// TIA Portal V15.1 export
// export: Created 2020-06-12T07:35:42.5849609Z, ExportSetting None, DisplayName Totally Integrated Automation Portal, DisplayVersion V15.1, DisplayName TIA Portal Openness, DisplayVersion V15.1, DisplayName STEP 7 Professional, DisplayVersion V15.1, DisplayName STEP 7 Safety, DisplayVersion V15.1, DisplayName WinCC Advanced, DisplayVersion V15.1
FUNCTION "CW_Module" : Void   // FC118, FBD
TITLE = CW Module (HC-lines cooling) handle
{ S7_Optimized_Access := 'TRUE' }
// stored: SetENOAutomatically False
   VAR_TEMP
      tStart_heater : Bool;
      tHeater_on : Bool;
      pump1_start : Bool;
      pump2_start : Bool;
      _heat_off : Real;
      tReqOn : Bool;
      tReqOff : Bool;
      tStage : Int;
      tFlowset : Real;
      tCVMin : Real;
      tCVMax : Real;
   END_VAR
   VAR_TEMP   // added for the SCL form of the ladder/FBD networks
      _w1 : Bool;
      _w2 : Bool;
   END_VAR
BEGIN

REGION Network 1: HMI request treat
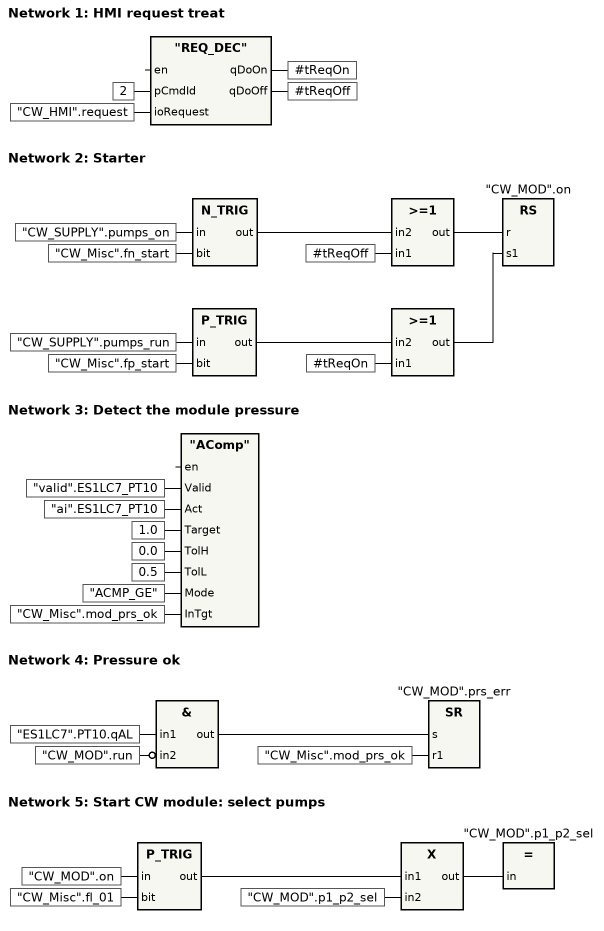
   "REQ_DEC"(pCmdId := 2, ioRequest := "CW_HMI".request, qDoOn => #tReqOn, qDoOff => #tReqOff);
END_REGION

REGION Network 2: Starter
   #_w1 := NOT "CW_SUPPLY".pumps_on AND "CW_Misc".fn_start;   // falling edge
   "CW_Misc".fn_start := "CW_SUPPLY".pumps_on;
   #_w2 := "CW_SUPPLY".pumps_run AND NOT "CW_Misc".fp_start;   // rising edge
   "CW_Misc".fp_start := "CW_SUPPLY".pumps_run;
   IF #_w1 OR #tReqOff THEN
       "CW_MOD".on := FALSE;   // RS flip-flop
   END_IF;
   IF #_w2 OR #tReqOn THEN "CW_MOD".on := TRUE; END_IF;
END_REGION

REGION Network 3: Detect the module pressure
   "AComp"(Valid := "valid".ES1LC7_PT10,
           Act := "ai".ES1LC7_PT10,
           Target := 1.0,
           TolH := 0.0,
           TolL := 0.5,
           Mode := "ACMP_GE",
           InTgt := "CW_Misc".mod_prs_ok);
END_REGION

REGION Network 4: Pressure ok
   // That is critical only before start
   IF "ES1LC7".PT10.qAL AND NOT "CW_MOD".run THEN
       "CW_MOD".prs_err := TRUE;   // SR flip-flop
   END_IF;
   IF "CW_Misc".mod_prs_ok THEN "CW_MOD".prs_err := FALSE; END_IF;
END_REGION

REGION Network 5: Start CW module: select pumps
   #_w1 := "CW_MOD".on AND NOT "CW_Misc".fl_01;   // rising edge
   "CW_Misc".fl_01 := "CW_MOD".on;
   "CW_MOD".p1_p2_sel := #_w1 XOR "CW_MOD".p1_p2_sel;
END_REGION

REGION Network 6: Module pumps LOCK
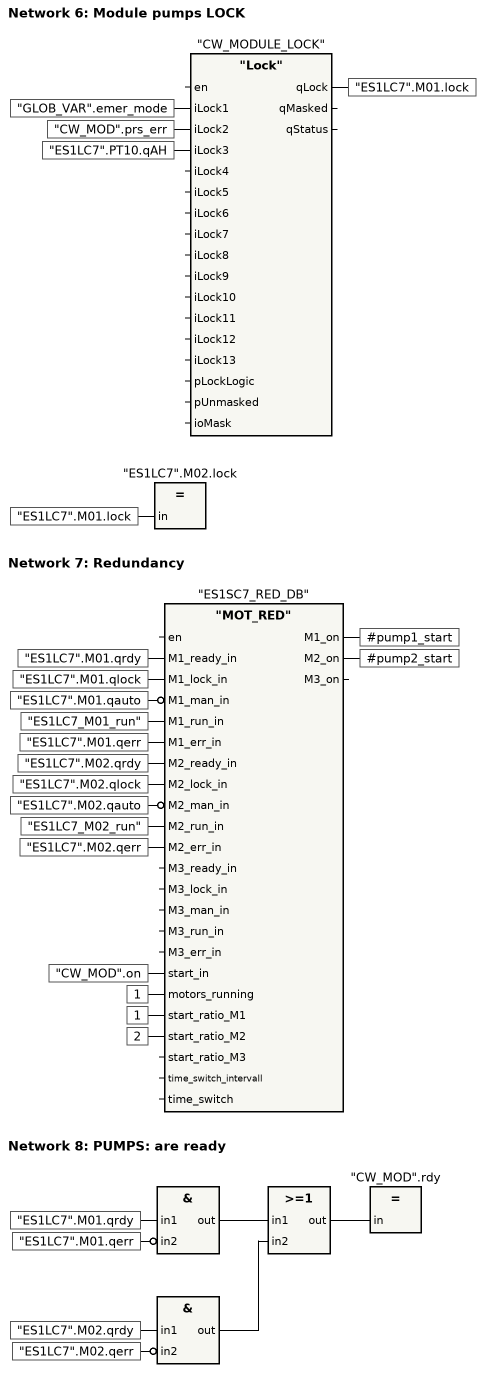
   "CW_MODULE_LOCK"(iLock1 := "GLOB_VAR".emer_mode,   // "Lock"
                    iLock2 := "CW_MOD".prs_err,
                    iLock3 := "ES1LC7".PT10.qAH,
                    qLock => "ES1LC7".M01.lock);
   "ES1LC7".M02.lock := "ES1LC7".M01.lock;
END_REGION

REGION Network 7: Redundancy
   "ES1SC7_RED_DB"(M1_ready_in := "ES1LC7".M01.qrdy,   // "MOT_RED"
                   M1_lock_in := "ES1LC7".M01.qlock,
                   M1_man_in := NOT "ES1LC7".M01.qauto,
                   M1_run_in := "ES1LC7_M01_run",
                   M1_err_in := "ES1LC7".M01.qerr,
                   M2_ready_in := "ES1LC7".M02.qrdy,
                   M2_lock_in := "ES1LC7".M02.qlock,
                   M2_man_in := NOT "ES1LC7".M02.qauto,
                   M2_run_in := "ES1LC7_M02_run",
                   M2_err_in := "ES1LC7".M02.qerr,
                   start_in := "CW_MOD".on,
                   motors_running := 1,
                   start_ratio_M1 := 1,
                   start_ratio_M2 := 2,
                   M1_on => #pump1_start,
                   M2_on => #pump2_start);
END_REGION

REGION Network 8: PUMPS: are ready
   "CW_MOD".rdy := ("ES1LC7".M01.qrdy AND NOT "ES1LC7".M01.qerr) OR ("ES1LC7".M02.qrdy AND NOT "ES1LC7".M02.qerr);
END_REGION

REGION Network 9: PUMPs: are(is) running
   // The stable running state is delayed for a ramp time.
   // In this case the ramp time is 50s, we take 60s.
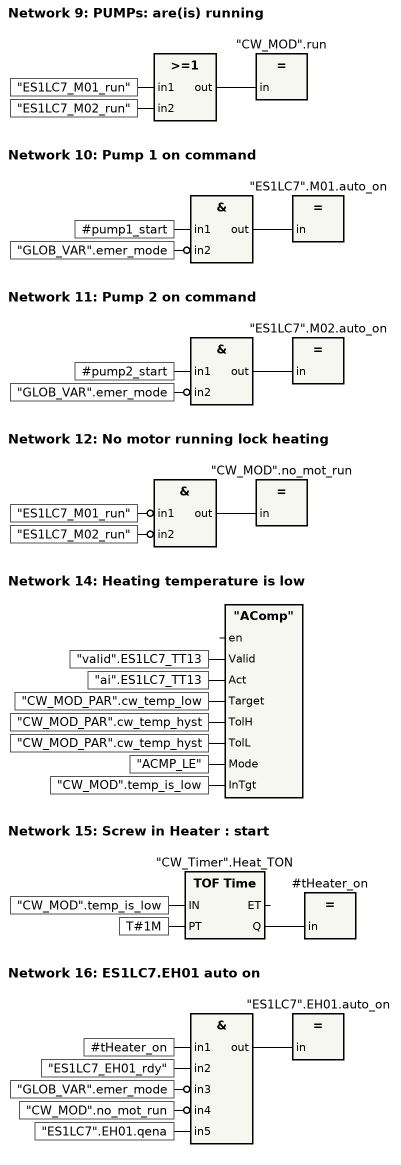
   "CW_MOD".run := "ES1LC7_M01_run" OR "ES1LC7_M02_run";
END_REGION

REGION Network 10: Pump 1 on command
   "ES1LC7".M01.auto_on := #pump1_start AND NOT "GLOB_VAR".emer_mode;
END_REGION

REGION Network 11: Pump 2 on command
   "ES1LC7".M02.auto_on := #pump2_start AND NOT "GLOB_VAR".emer_mode;
END_REGION

REGION Network 12: No motor running lock heating
   "CW_MOD".no_mot_run := NOT "ES1LC7_M01_run" AND NOT "ES1LC7_M02_run";
END_REGION

REGION Network 13: [Heating/Recooling]
END_REGION

REGION Network 14: Heating temperature is low
   "AComp"(Valid := "valid".ES1LC7_TT13,
           Act := "ai".ES1LC7_TT13,
           Target := "CW_MOD_PAR".cw_temp_low,
           TolH := "CW_MOD_PAR".cw_temp_hyst,
           TolL := "CW_MOD_PAR".cw_temp_hyst,
           Mode := "ACMP_LE",
           InTgt := "CW_MOD".temp_is_low);
END_REGION

REGION Network 15: Screw in Heater : start
   "CW_Timer".Heat_TON.TOF(IN := "CW_MOD".temp_is_low, PT := T#1M);
   #tHeater_on := "CW_Timer".Heat_TON.Q;
END_REGION

REGION Network 16: ES1LC7.EH01 auto on
   "ES1LC7".EH01.auto_on := #tHeater_on AND "ES1LC7_EH01_rdy" AND NOT "GLOB_VAR".emer_mode AND NOT "CW_MOD".no_mot_run AND "ES1LC7".EH01.qena;
END_REGION

REGION Network 17: ES1LC7.EH01 Lock
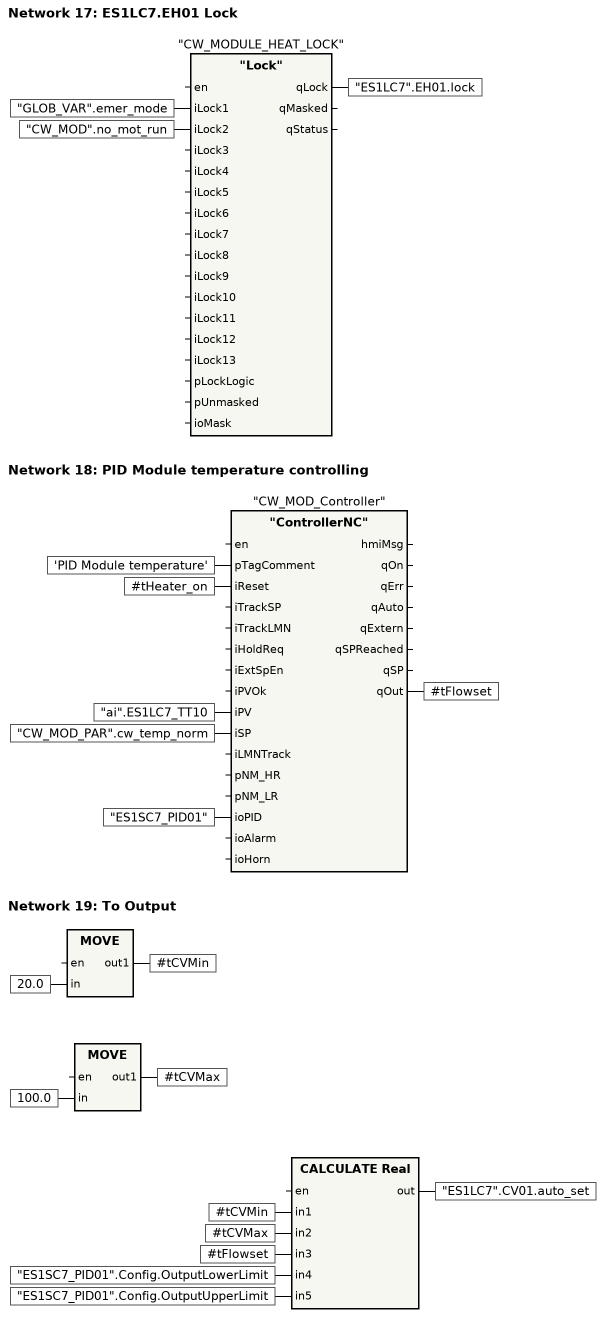
   "CW_MODULE_HEAT_LOCK"(iLock1 := "GLOB_VAR".emer_mode,   // "Lock"
                         iLock2 := "CW_MOD".no_mot_run,
                         qLock => "ES1LC7".EH01.lock);
END_REGION

REGION Network 18: PID Module temperature controlling
   "CW_MOD_Controller"(pTagComment := 'PID Module temperature',   // "ControllerNC"
                       iReset := #tHeater_on,
                       iPV := "ai".ES1LC7_TT10,
                       iSP := "CW_MOD_PAR".cw_temp_norm,
                       ioPID := "ES1SC7_PID01",
                       qOut => #tFlowset);
END_REGION

REGION Network 19: To Output
   // That is not good idea to fully close CV
   #tCVMin := 20.0;
   #tCVMax := 100.0;
   "ES1LC7".CV01.auto_set := #tCVMax - (#tCVMin + (#tCVMax - #tCVMin) * ((#tFlowset - "ES1SC7_PID01".Config.OutputLowerLimit) / ("ES1SC7_PID01".Config.OutputUpperLimit - "ES1SC7_PID01".Config.OutputLowerLimit)));
END_REGION

REGION Network 20: Enable Alarm
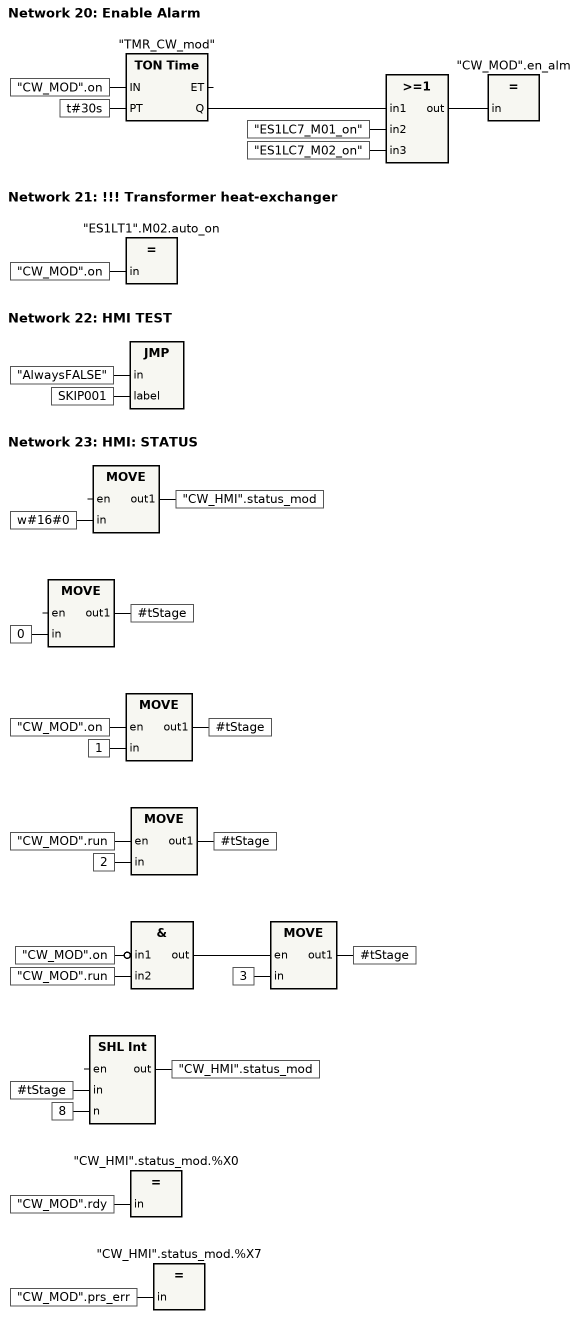
   "TMR_CW_mod".TON(IN := "CW_MOD".on, PT := t#30s);
   "CW_MOD".en_alm := "TMR_CW_mod".Q OR "ES1LC7_M01_on" OR "ES1LC7_M02_on";
END_REGION

REGION Network 21: !!! Transformer heat-exchanger
   "ES1LT1".M02.auto_on := "CW_MOD".on;
END_REGION

REGION Network 22: HMI TEST
   // This network is used for HMI test
   IF "AlwaysFALSE" THEN GOTO SKIP001; END_IF;
END_REGION

REGION Network 23: HMI: STATUS
   "CW_HMI".status_mod := w#16#0;
   #tStage := 0;
   IF "CW_MOD".on THEN #tStage := 1; END_IF;
   IF "CW_MOD".run THEN #tStage := 2; END_IF;
   IF NOT "CW_MOD".on AND "CW_MOD".run THEN #tStage := 3; END_IF;
   "CW_HMI".status_mod := SHL(IN := #tStage, N := 8);
   "CW_HMI".status_mod.%X0 := "CW_MOD".rdy;
   "CW_HMI".status_mod.%X7 := "CW_MOD".prs_err;
END_REGION

REGION Network 24
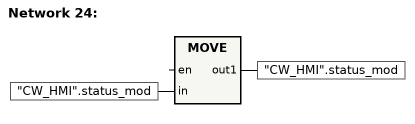
   SKIP001:
   "CW_HMI".status_mod := "CW_HMI".status_mod;
END_REGION
END_FUNCTION
